FUNCTION_BLOCK FB_Moto EXTENDS FB_Vehiculo
VAR_INPUT
	aceleracion : REAL;
END_VAR
VAR_OUTPUT
END_VAR
VAR
END_VAR

METHOD getAceleracion : REAL
VAR_INPUT
END_VAR
getAceleracion := aceleracion;
END_METHOD

END_FUNCTION_BLOCK

(* stored: Version 1.1.0.1, ProductVersion 3.1.4024.12
   POU FB_Moto: Id {2cd26c6e-3eb4-49c2-aa2c-988956508106}, SpecialFunc None
   Method getAceleracion: Id {8234eae8-cfda-499b-9f77-a929ee25ba05} *)
